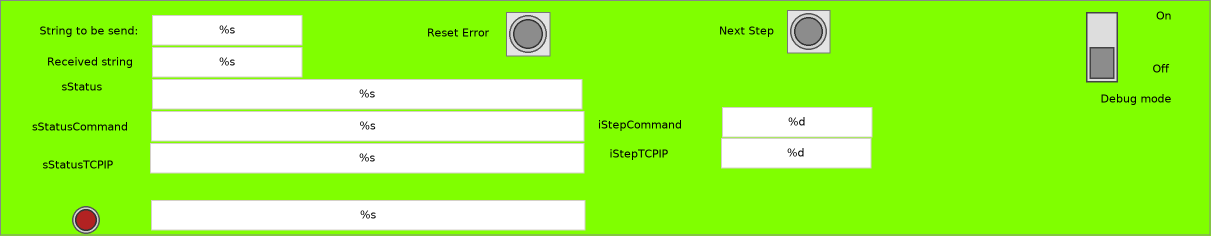
VISUALIZATION HMI  // 1211x236
    Label (14,16 150x30), "String to be send:"
    Label (15,47 150x30), "Received string"
    Textfield (152,15 150x30), "%s", text variable: Visu.visuStingToBeSent
    Textfield (152,47 150x30), "%s", text variable: Visu.visuReceivedString
    Label (7,72 150x30), "sStatus"
    Label (5,112 150x30), "sStatusCommand"
    Label (3,150 150x30), "sStatusTCPIP"
    Label (565,110 150x30), "iStepCommand"
    Textfield (152,79 430x30), "%s", text variable: Visu.visuStatus
    Label (564,139 150x30), "iStepTCPIP"
    Textfield (151,111 433x30), "%s", text variable: Visu.visuStatusCommand
    Textfield (722,107 150x30), "%d", text variable: Visu.visuStepCommand
    Textfield (721,138 150x30), "%d", text variable: Visu.visuStepTCPIP
    Textfield (150,143 434x30), "%s", text variable: Visu.visuStatusTCPIP
    Textfield (151,200 434x30), "%s", text variable: Main.IV3.sERROR
    Lamp1 (70,204 32x32), variable: Main.IV3.bERROR, style: Lamp-Lamp1-Red
    Group (1061,1 150x113)
        DipSwitch (6,11 70x70), variable: Main.IV3.bDebugModeOn, behaviour: TOGGLE, style: Switch-DipSwitch-Gray
        Rectangle (0,83 150x30), "Debug mode"
        Rectangle (75,0 56x30), "On"
        Rectangle (72,53 56x30), "Off"
    PushSwitch (506,9 44x50), variable: MAIN.IV3.bResetERROR, behaviour: TOGGLE, style: Switch-PushSwitch-Gray
    Label (418,18 80x30), "Reset Error"
    PushSwitch (787,10 43x43), variable: MAIN.IV3.bStepButton, behaviour: TOGGLE, style: Switch-PushSwitch-Gray
    Label (699,16 78x30), "Next Step"
END_VISUALIZATION

(* stored: Version 1.1.0.1, ProductVersion 3.1.4024.14
   Visu HMI: Id {1d227db8-b5b9-4ede-ae67-6cd7ce29c1d9} *)
